// Mitsubishi GX Works2 project: hung_creat_plc_dich_bit   PLC: FX3U/FX3UC

PROGRAM MAIN
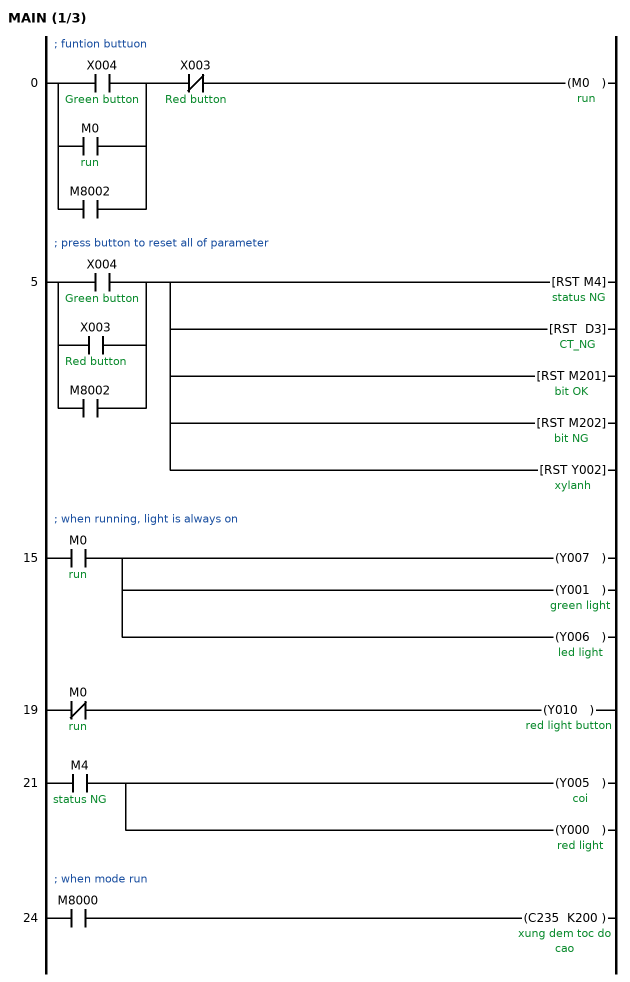
; funtion buttuon
0     LD      X004  ; Green button
      OR      M0  ; run
      OR      M8002
      ANI     X003  ; Red button
      OUT     M0  ; run
; press button to reset all of parameter
5     LD      X004  ; Green button
      OR      X003  ; Red button
      OR      M8002
      RST     M4  ; status NG
      RST     D3  ; CT_NG
      RST     M201  ; bit OK
      RST     M202  ; bit NG
      RST     Y002  ; xylanh
; when running, light is always on
15    LD      M0  ; run
      OUT     Y007
      OUT     Y001  ; green light
      OUT     Y006  ; led light
19    LDI     M0  ; run
      OUT     Y010  ; red light button
21    LD      M4  ; status NG
      OUT     Y005  ; coi
      OUT     Y000  ; red light
; when mode run
24    LD      M8000
      OUT     C235 K200  ; xung dem toc do  cao
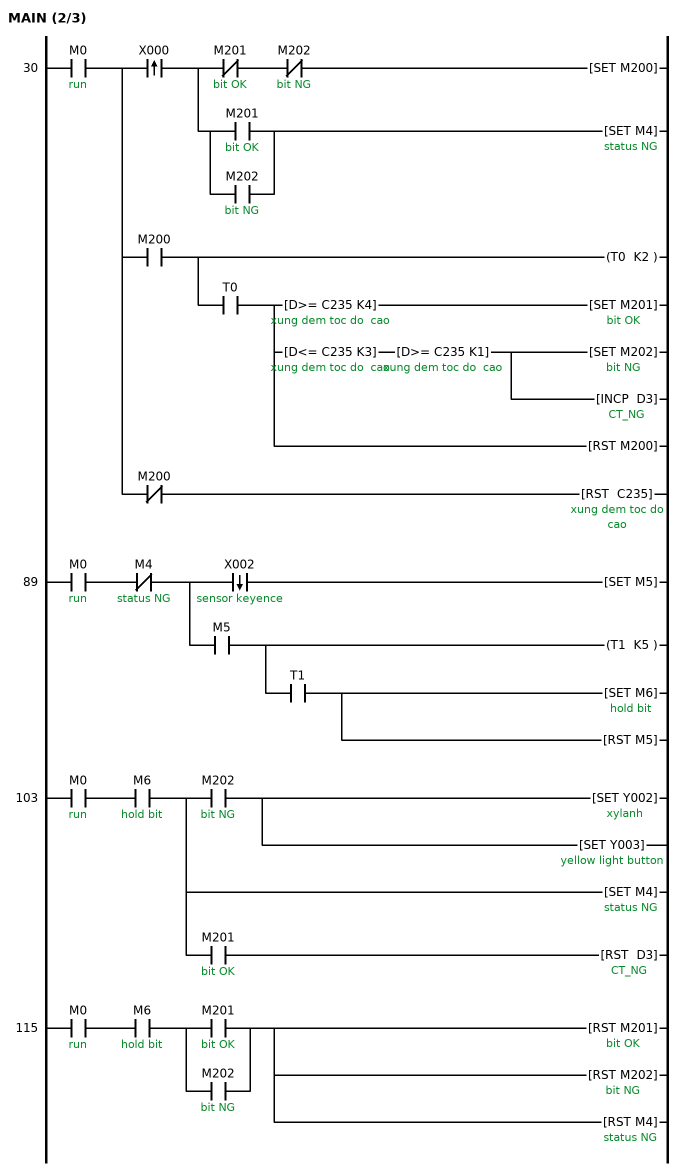
30    LD      M0  ; run
      MPS
      ANDP    X000
      MPS
      ANI     M201  ; bit OK
      ANI     M202  ; bit NG
      SET     M200
      MPP
      LD      M201  ; bit OK
      OR      M202  ; bit NG
      ANB
      SET     M4  ; status NG
      MRD
      AND     M200
      OUT     T0 K2
      AND     T0
      MPS
      ANDD>=  C235 K4  ; xung dem toc do  cao
      SET     M201  ; bit OK
      MRD
      ANDD<=  C235 K3  ; xung dem toc do  cao
      ANDD>=  C235 K1  ; xung dem toc do  cao
      SET     M202  ; bit NG
      INCP    D3
      MPP
      RST     M200
      MPP
      ANI     M200
      RST     C235  ; xung dem toc do  cao
89    LD      M0  ; run
      ANI     M4  ; status NG
      MPS
      ANDF    X002  ; sensor keyence
      SET     M5
      MPP
      AND     M5
      OUT     T1 K5
      AND     T1
      SET     M6  ; hold bit
      RST     M5
103   LD      M0  ; run
      AND     M6  ; hold bit
      MPS
      AND     M202  ; bit NG
      SET     Y002  ; xylanh
      SET     Y003  ; yellow light button
      MPP
      SET     M4  ; status NG
      AND     M201  ; bit OK
      RST     D3  ; CT_NG
115   LD      M0  ; run
      AND     M6  ; hold bit
      LD      M201  ; bit OK
      OR      M202  ; bit NG
      ANB
      RST     M201  ; bit OK
      RST     M202  ; bit NG
      RST     M4  ; status NG
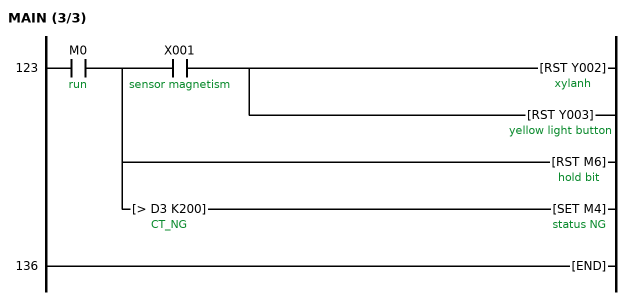
123   LD      M0  ; run
      MPS
      AND     X001  ; sensor magnetism
      RST     Y002  ; xylanh
      RST     Y003  ; yellow light button
      MPP
      RST     M6  ; hold bit
      AND>    D3 K200  ; CT_NG
      SET     M4  ; status NG
136   END
END_PROGRAM

// device comments not shown above
D0  ; CT
M3  ; bit reset NG and OK
